(*
SPDX-FileCopyrightText: © 2026 Oleksandr Tiutyk <trofimich@gmail.com>
SPDX-License-Identifier: MIT
License: https://opensource.org/license/mit
*)

(*!
<summary>
Sample workflow exposing corner movement flags, current X/Y position and control commands for visualization.
</summary>
*)

{attribute 'no_explicit_call' := 'do not call this function block directly'}
{attribute 'enable_dynamic_creation'}
FUNCTION_BLOCK DemoWorkflow EXTENDS TOF_Workflow.Workflow
VAR_INPUT
	StartOrResumeRequest : BOOL;
	SuspendRequest : BOOL;
	CancelRequest : BOOL;
	ResetRequest : BOOL;
	
	MoveFrom1To2 : BOOL;
	MoveFrom2To3 : BOOL;	
	MoveFrom3To4 : BOOL;	
	MoveFrom4To1 : BOOL;
END_VAR
VAR_OUTPUT	
	XPosition : INT;
	YPosition : INT;

	StateName : STRING(20);
END_VAR
VAR_STAT
	{attribute 'hide'} 
	_WorkflowClassName : STRING := __POUNAME();
END_VAR

(*!
<summary>Gets the runtime class name of this object.</summary>
<description>Returns initialized static storage without reading derived instance state.</description>
*)
{attribute 'monitoring' := 'call'}
PROPERTY ClassName : REFERENCE TO STRING
GET
ClassName REF= _WorkflowClassName;
END_GET
END_PROPERTY

(*!
<summary>Registers the six workflow variables used by the sample activities.</summary>
*)
METHOD PROTECTED InitializeVariables
BindPlcVariable(name := 'XPosition', plcVariable := XPosition);
BindPlcVariable(name := 'YPosition', plcVariable := YPosition);

BindPlcVariable(name := 'MoveFrom1To2', plcVariable := MoveFrom1To2);
BindPlcVariable(name := 'MoveFrom2To3', plcVariable := MoveFrom2To3);
BindPlcVariable(name := 'MoveFrom3To4', plcVariable := MoveFrom3To4);
BindPlcVariable(name := 'MoveFrom4To1', plcVariable := MoveFrom4To1);
END_METHOD

METHOD FB_init : BOOL
VAR_INPUT
	bInitRetains : BOOL; // TRUE: the retain variables are initialized (reset warm / reset cold)
	bInCopyCode : BOOL;  // TRUE: the instance will be copied to the copy code afterward (online change)
END_VAR
Name := "Demo workflow";
END_METHOD

(*!
<summary>Gets the namespace name of this object.</summary>
*)
{attribute 'monitoring' := 'call'}
PROPERTY NamespaceName : REFERENCE TO STRING
GET
NamespaceName REF= CurrentNamespace.Name;
END_GET
END_PROPERTY

(*!
<summary>Updates the formatted StateName output after each cyclic execution step.</summary>
*)
METHOD PROTECTED OnAfterRootActivityExecute
StateName := TO_STRING(State);

TOF_Core.Strings.ReplaceInSource255(sourceString := StateName, oldSubstring := 'ACTIVE_', newSubstring := '');
TOF_Core.Strings.ReplaceInSource255(sourceString := StateName, oldSubstring := 'PASSIVE_', newSubstring := '');
END_METHOD

(*!
<summary>Processes pending user command flags before RootActivity.Execute runs.</summary>
*)
METHOD PROTECTED OnBeforeRootActivityExecute
IF CancelRequest THEN
	RequestCancel(reason := "Cancelled by user");
ELSIF SuspendRequest THEN
	RequestSuspend();
ELSIF ResetRequest THEN
	RequestReset();
ELSIF StartOrResumeRequest THEN
	RequestStart();
END_IF

CancelRequest := FALSE;
SuspendRequest := FALSE;
ResetRequest := FALSE;
StartOrResumeRequest := FALSE;
END_METHOD

(*!
<summary>Resets XPosition and YPosition to the origin when resetting the workflow.</summary>
<param name="abortRequest">Set TRUE to cancel the reset request.</param>
*)
METHOD PROTECTED OnRootActivityRequestReset
VAR_OUTPUT
	abortRequest : BOOL;
END_VAR
XPosition := 0;
YPosition := 0;
END_METHOD

(*!
<summary>Resets XPosition and YPosition to the origin when starting a fresh run from PASSIVE_READY.</summary>
<param name="abortRequest">Set TRUE to cancel the start request.</param>
*)
METHOD PROTECTED OnRootActivityRequestStart
VAR_OUTPUT
	abortRequest : BOOL;
END_VAR
VAR
	currentRootActivity : TOF_Workflow.IActivity;
END_VAR
currentRootActivity := RootActivity;

IF currentRootActivity <> 0
	AND_THEN currentRootActivity.State <> TOF_Workflow.WORKFLOW_ELEMENT_STATE.PASSIVE_SUSPENDED
THEN
	XPosition := 0;
	YPosition := 0;
END_IF
END_METHOD

(*!
<summary>Gets the size in bytes of this function block instance.</summary>
*)
{attribute 'monitoring' := 'call'}
PROPERTY SelfSize : ULINT
GET
SelfSize := XSIZEOF(THIS^);
END_GET
END_PROPERTY

END_FUNCTION_BLOCK

(* stored: Version 1.1.0.1
   POU DemoWorkflow: Id {78bf3e61-8572-48b3-a515-1429d4fe5b8c}, SpecialFunc None
   Folder Overriden members: Id {e1bd6d81-733a-4b2d-8159-643d9dc52551}
   Property ClassName: Id {b5279f96-3cc0-4b10-94f1-c41eea8241ef}
   Get Get: Id {d0b1f1e5-44e8-44bf-afb9-34b1f18937f7}
   Method InitializeVariables: Id {51b26f57-2957-4301-a216-0f399dc62fe6}
   Method FB_init: Id {2ac10e27-5c07-430f-8815-6a49562c7896}
   Property NamespaceName: Id {6857a071-d211-497a-8b1d-17675e8ef5ee}
   Get Get: Id {362b15c6-d806-46db-b10d-07897f4d3323}
   Method OnAfterRootActivityExecute: Id {b3012c22-5e10-4343-868e-37d17a14cf5d}
   Method OnBeforeRootActivityExecute: Id {2559e0ca-4ccd-4369-93ae-b8b12073eddc}
   Method OnRootActivityRequestReset: Id {8f4a21c3-6d18-4b75-9a2e-3c7150e8d491}
   Method OnRootActivityRequestStart: Id {db98a397-a185-4880-ae49-598e0c480c81}
   Property SelfSize: Id {5b4d1388-29da-418f-aee0-1a2a0c82dc24}
   Get Get: Id {bebd553c-a106-43a4-afc0-d3e65361e96a} *)
